// TIA Portal V20 export
TYPE "CBS_Datos_config"
   STRUCT
      Numero_MesaAsociada : UInt;   // Numero de Mesa Asociado al Quimarox
      Numero_vagones : Int;
      ConfigEvento : Struct
         SSCC : Bool;
      END_STRUCT;
      Long_Vagon_mm : Int;
      Long_Util_vagon_mm : Int;
      dist_ini_vag_a_phs_mm : Int;
      maximo_encoder : DInt;
      relacion_mm_pulso : Real;
      DatosTrabajo : Struct
         Memoria_Dato_Encoder : DInt;
         Hora_Ultimo_Refresco : Time_Of_Day;
         Hora_Anterior_Refresco : Time_Of_Day;
         Memoria_MCKEY : UDInt;
         Actualizar_Config : Bool;
         Memoria_Inicializacion : Bool;
         Memoria_Actualizacion_Config : Bool;
         Error_Referenciacion : Bool;
         Error_Timeout_Com_SAC : Bool;
      END_STRUCT;
   END_STRUCT;
END_TYPE
